PROGRAM P_Demo_F_BYTE
VAR
    nStatusByte   : BYTE := 16#A5; // 业务量（BYTE）
    bPackArg      : BOOL; // 在线置 TRUE 触发一次打包
    argDescriptor : T_Arg; // 打包后的 T_Arg 描述符（含 eType/cbLen/pData）
END_VAR

// ============================================================
// Tc2_Utilities.F_BYTE 演示程序（FUNCTION，返回 T_Arg）
// ============================================================
// 场景：把 BYTE 业务量打包为 T_Arg，供下游 EventLogger / FormatString2
//       / ADS 消息的可变参数机制使用。
// 价值：替代手填 T_Arg 三字段（eType/cbLen/pData），一行调用搞定。
// 验证：在线写 nStatusByte 为示例值，bPackArg := TRUE；
//       下一周期 argDescriptor.cbLen = SIZEOF(BYTE)，argDescriptor.pData <> 0。
// ============================================================

IF bPackArg THEN
    // 单次完整调用：返回的 T_Arg 立即可喂给 F_PutInArg(arg := argDescriptor, ...)
    argDescriptor := F_BYTE(nStatusByte);
    bPackArg := FALSE;
END_IF;

END_PROGRAM

(* stored: Version 1.1.0.1, ProductVersion 3.1.4024.5
   POU P_Demo_F_BYTE: Id {e64654ad-a6b3-5602-8c85-c3e3495718cc}, SpecialFunc None *)
